(* Schneider Machine Expert - Basic project Exercise-21-Alarm System of any Company, file version 2.9.0.0 *)
(* ProjectInformations: Name=New project *)

HARDWARE
  Cpu 0: TM221C24R
  EthernetConfiguration: NetworkName=M221, IpAllocationMode=FixedAddress, IpAddress=0.0.0.0, SubnetMask=0.0.0.0
  SerialLineConfiguration: Baud=Baud19200, Parity=ParityEven, DataBits=DataBits8, StopBits=StopBits1, PhysicalMedium=PhysicalMediumRs485, SlaveId=1, Addressing=SlaveAddressing
  MastTask: UsePeriodScanMode=false, PeriodScan=100
  FastTask: Period=255
  CpuBehavior: StartingMode=StartAsPreviousState, AutoSaveRamOnEeprom=true, WatchdogPeriod=250

SYMBOLS  (address, symbol, comment, settings)
  %I0.0     SWITCH_1
  %I0.1     SWITCH_2
  %I0.2     SWITCH_3
  %I0.3     SWITCH_4
  %I0.4     SWITCH_5
  %I0.5     SWITCH_6
  %I0.6     SWITCH_7
  %I0.7     SWITCH_8
  %Q0.0     ALARM

POU New POU
  (* SectionNumber=1 *)

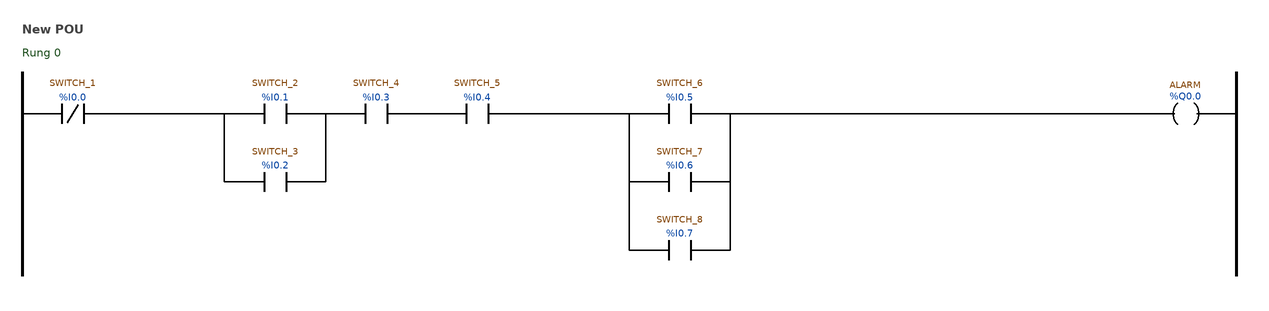

// Rung 0
  LDN %I0.0               (* SWITCH_1 *)
  AND( %I0.1              (* SWITCH_2 *)
  OR %I0.2                (* SWITCH_3 *)
  )
  AND %I0.3               (* SWITCH_4 *)
  AND %I0.4               (* SWITCH_5 *)
  AND( %I0.5              (* SWITCH_6 *)
  OR %I0.6                (* SWITCH_7 *)
  OR %I0.7                (* SWITCH_8 *)
  )
  ST %Q0.0                (* ALARM *)
  // as ST:
  //   ALARM := NOT SWITCH_1 AND (SWITCH_2 OR SWITCH_3) AND SWITCH_4 AND SWITCH_5 AND (SWITCH_6 OR SWITCH_7 OR SWITCH_8);
